(* PLC project SafeLOGIC-1, BrAutomation SafeDESIGNER  4.3.2.11 *)
(* stored: companyURL http://www.br-automation.com, creationDateTime Thu May 17 17:30:16 2018 *)

PROGRAM ScaleSAFEINT

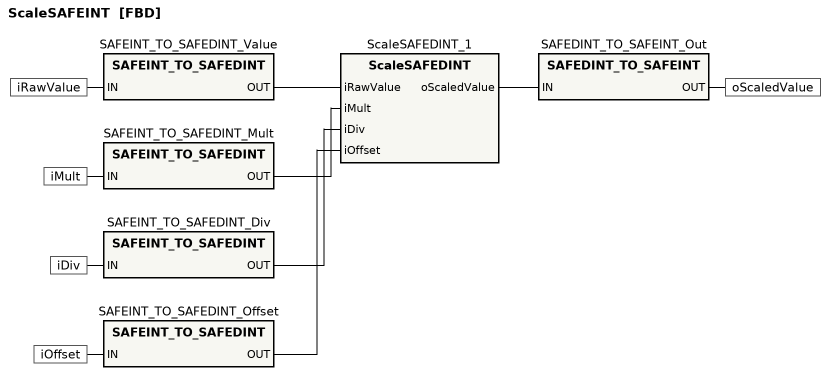
(* FBD diagram, written out as Structured Text *)
SAFEINT_TO_SAFEDINT_Value(IN := iRawValue);
SAFEINT_TO_SAFEDINT_Mult(IN := iMult);
SAFEINT_TO_SAFEDINT_Div(IN := iDiv);
SAFEINT_TO_SAFEDINT_Offset(IN := iOffset);
ScaleSAFEDINT_1(iRawValue := SAFEINT_TO_SAFEDINT_Value.OUT, iMult := SAFEINT_TO_SAFEDINT_Mult.OUT, iDiv := SAFEINT_TO_SAFEDINT_Div.OUT, iOffset := SAFEINT_TO_SAFEDINT_Offset.OUT);
SAFEDINT_TO_SAFEINT_Out(IN := ScaleSAFEDINT_1.oScaledValue);
oScaledValue := SAFEDINT_TO_SAFEINT_Out.OUT;
END_PROGRAM
